PROGRAM Demo
VAR

    fbMotionLogger : FB_MotionLogger;
    // Persistant storage
    fbPersistentDataStorage : FB_PersistentDataStorage;
    M1 : ST_MotionEpicsInterface;

    fbMotionStage : FB_MotionStageNC(	sName := 'NC',
                                        stMotionEpicsItf := M1,
                                        AxisRef := NcAxis_GVL.NC,
                                        iMotionLogger := fbMotionLogger,
                                        iPersistentDataStorage := fbPersistentDataStorage
                                    ) := (	HardwareEnable:=TRUE,
                                            UserEnable:=TRUE,
                                            LimBackward := TRUE,
                                            LimForward:=TRUE,
                                            BrakeMode := E_StageBrakeMode.IF_MOVING,
                                            EnableMode:=ENUM_StageEnableMode.DURING_MOTION,
                                            HomeMode:=E_EpicsHomeCmd.ABSOLUTE_SET
                                    );
END_VAR

fbMotionLogger();
fbPersistentDataStorage();
fbMotionStage();

END_PROGRAM

(* stored: Version 1.1.0.1
   POU Demo: Id {61c6dfbc-a7dc-4c03-9ea3-aa217d748554}, SpecialFunc None *)
